{attribute addProperty BoxType "EP3314-0002-0018"}
{attribute addProperty Id "StatusAT %I*Status_7401E3071621ValueAT %I*INT16217"}
{attribute addProperty CRC "1073525614"}
{attribute addProperty SizeInBites "32"}
{attribute addProperty SizeInBytes "4"}
TYPE TC_TCInputs_Channel_3FFCB36E :
STRUCT
	{attribute addProperty Name "Status"}
	Status AT %I* : Status_7401E307;
	{attribute addProperty Name "Value"}
	Value AT %I* : INT;
END_STRUCT
END_TYPE

(* stored: Version 1.2.0.0, ProductVersion 3.1.4024.9
   DUT TC_TCInputs_Channel_3FFCB36E: Id {8bedcf75-3294-4b5a-b3bb-faf98401f617} *)
